// TIA Portal V20 export
FUNCTION_BLOCK "Lift"   // FB8, LAD
{ S7_Optimized_Access := 'TRUE' }
// stored: MemoryReserve 100, SetENOAutomatically false
   VAR
      Lift_Driver { S7_SetPoint := 'True'} : "Lift_Driver";
      Lift_Drive_To_Level { S7_SetPoint := 'True'} : "Lift_Drive_To_Level";
      Forward_Auto { S7_SetPoint := 'True'} : Bool;
      Backward_Auto : Bool;
      Velocity : LReal;
      Reset : Bool;
      Halt_Auto : Bool;
      Power_Auto : Bool;
   END_VAR
BEGIN

REGION Network 1
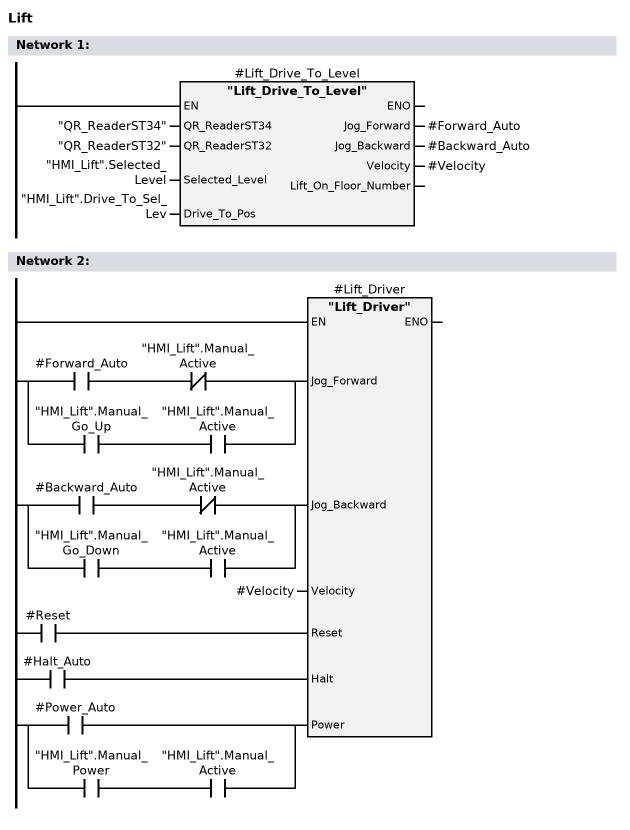
   RUNG wire#powerrail
      #Lift_Drive_To_Level(QR_ReaderST34 := "QR_ReaderST34", QR_ReaderST32 := "QR_ReaderST32", Selected_Level := "HMI_Lift".Selected_Level, Drive_To_Pos := "HMI_Lift".Drive_To_Sel_Lev, Jog_Forward => #Forward_Auto, Jog_Backward => #Backward_Auto, Velocity => #Velocity, Lift_On_Floor_Number =>)
   END_RUNG
   // the same network as SCL:
   #Lift_Drive_To_Level(QR_ReaderST34 := "QR_ReaderST34",   // "Lift_Drive_To_Level"
                        QR_ReaderST32 := "QR_ReaderST32",
                        Selected_Level := "HMI_Lift".Selected_Level,
                        Drive_To_Pos := "HMI_Lift".Drive_To_Sel_Lev,
                        Jog_Forward => #Forward_Auto,
                        Jog_Backward => #Backward_Auto,
                        Velocity => #Velocity);
END_REGION

REGION Network 2
   RUNG wire#powerrail
      #Lift_Driver(Jog_Forward := wire#w1, Jog_Backward := wire#w2, Reset := wire#w3, Halt := wire#w4, Power := wire#w5, Velocity := #Velocity)
   END_RUNG
   RUNG wire#powerrail
      Contact( #Forward_Auto )
      I_Contact( "HMI_Lift".Manual_Active )
   END_RUNG wire#w1
   RUNG wire#powerrail
      Contact( "HMI_Lift".Manual_Go_Up )
      Contact( "HMI_Lift".Manual_Active )
   END_RUNG wire#w1
   RUNG wire#powerrail
      Contact( #Backward_Auto )
      I_Contact( "HMI_Lift".Manual_Active )
   END_RUNG wire#w2
   RUNG wire#powerrail
      Contact( "HMI_Lift".Manual_Go_Down )
      Contact( "HMI_Lift".Manual_Active )
   END_RUNG wire#w2
   RUNG wire#powerrail
      Contact( #Reset )
   END_RUNG wire#w3
   RUNG wire#powerrail
      Contact( #Halt_Auto )
   END_RUNG wire#w4
   RUNG wire#powerrail
      Contact( #Power_Auto )
   END_RUNG wire#w5
   RUNG wire#powerrail
      Contact( "HMI_Lift".Manual_Power )
      Contact( "HMI_Lift".Manual_Active )
   END_RUNG wire#w5
   // the same network as SCL:
   #Lift_Driver(Jog_Forward := (#Forward_Auto AND NOT "HMI_Lift".Manual_Active) OR ("HMI_Lift".Manual_Go_Up AND "HMI_Lift".Manual_Active),   // "Lift_Driver"
                Jog_Backward := (#Backward_Auto AND NOT "HMI_Lift".Manual_Active) OR ("HMI_Lift".Manual_Go_Down AND "HMI_Lift".Manual_Active),
                Velocity := #Velocity,
                Reset := #Reset,
                Halt := #Halt_Auto,
                Power := #Power_Auto OR ("HMI_Lift".Manual_Power AND "HMI_Lift".Manual_Active));
END_REGION
END_FUNCTION_BLOCK
